FUNCTION_BLOCK Forces6
VAR_INPUT
END_VAR
VAR_OUTPUT
END_VAR
VAR
END_VAR

END_FUNCTION_BLOCK

(* stored: Version 1.1.0.1, ProductVersion 3.1.4024.11
   POU Forces6: Id {c412c0a2-882b-4d65-a447-e77bb63c950b}, SpecialFunc None *)
